# EPICS autosave request: iocBoot/iocTune/auto_settings_tuneBO.req
file "tune_settings.req",                  P=$(P),  R=$(R)
file "tuneBO_settings.req",                P=$(P),  R=$(R)
